# EPICS alarm handler configuration: mps_database/bare/alarms/areas/mpln_l0b_mp04.alhConfig
GROUP NULL MPLN:L0B:MP04:1
$ALIAS MPS Link Node 54
$GUIDANCE
LTUH MPS
   Group Name: MPLN:L0B:MP04:1
   Summary PV:  MPLN:L0B:MP04:1:STATSUMY
$END
CHANNEL  MPLN:L0B:MP04:1    MPLN:L0B:MP04:1:MPS_EN_RBV		-----
CHANNEL  MPLN:L0B:MP04:1    MPLN:L0B:MP04:1:LC1_MODE_RBV		-----
